PROGRAM MAIN
VAR
	dtTimestamp : DATE_AND_TIME := DT#2017-04-04-12:42:42;
  	(* JSON document *)
  	fbJson			: FB_JsonSaxWriter;
	fbJsonDataType	: FB_JsonReadWriteDataType;
	sJsonDoc		: STRING(255); // Small JSON document, can be generated via GetDocument() for up to 255 characters
	sJsonDoc2		: STRING(2000); // Large JSON document, can be generated via CopyDocument()
	stValues		: ST_Values;
END_VAR

fbJson.ResetDocument();
fbJson.StartObject();
fbjson.AddKeyDateTime('Timestamp', dtTimestamp);
fbJsonDataType.AddJsonKeyValueFromSymbol(fbJson, 'Values', 'ST_Values', SIZEOF(stValues), ADR(stValues));
fbJsonDataType.AddJsonKeyPropertiesFromSymbol(fbJson, 'MetaData', 'ST_Values', 'Unit|DisplayName');
fbJson.EndObject();

sJsonDoc := fbJson.GetDocument();
fbJson.CopyDocument(sJsonDoc2, SIZEOF(sJsonDoc2));

END_PROGRAM

(* stored: Version 1.1.0.1, ProductVersion 3.1.4021.12
   POU MAIN: Id {ecb079e9-f108-4a4a-ab17-1dc515e9a429}, SpecialFunc None *)
